(* CODESYS project Step.project
   Title: Step
   Version: 0.0.0.0
   Author: MustafaZahid

Project tree, tasks and I/O mapping:
  MyController : TM241C24T/U, Schneider Electric, order no. TM241C24T/U, version 4.0.6.18
    application Application
      task MAST (cyclic, interval 20 ms, priority 15, watchdog 100 ms x 1) calls POU
      global variables GVL
      program POU [LD]
    DI : Digital Inputs, Schneider Electric, version 4.0.6.18
        input  iwDI_IW0 : WORD  // IW0
        input  ibDI_IB1 : BYTE  // IB1
    DQ : Digital Outputs, Schneider Electric, version 4.0.6.18
        settings: Outputs Usage = 3
        output qwDQ_QW0 : WORD  // QW0
        output qbDQ_QB1 : BYTE  // QB1
    Counters : Counters, Schneider Electric, version 4.0.6.18
    Pulse_Generators : Pulse Generators, Schneider Electric, version 4.0.6.18
        settings: Instance name = 'Axis_1'; B output History = 'old=-1 new=1'; A output History = 'old=-1 new=0'; Temporary Instance name = 'Axis_1'
    Cartridge_1 : Cartridge, Schneider Electric, version 4.0.6.18
    IO_Bus : IO bus - TM3, Schneider Electric, version 4.0.6.18
    COM_Bus : COM bus, Schneider Electric, version 4.0.6.18
    Serial_Line_1 : Serial line, Schneider Electric, version 4.0.6.18
      SoMachine_Network_Manager : SoMachine-Network Manager, Schneider Electric, version 4.0.0.2
    Serial_Line_2 : Serial line, Schneider Electric, version 4.0.6.18
      Modbus_Manager : Modbus Manager, Schneider Electric, version 4.0.0.2
*)

// MyController/Application/GVL
VAR_GLOBAL
END_VAR

// MyController/Application/POU
PROGRAM POU
VAR
	MC_Power: MC_Power_PTO;
	MC_MoveVelocity: MC_MoveVelocity_PTO;
	MC_Reset: MC_Reset_PTO;
	Power: BOOL;
	Start: BOOL;
	Reset: BOOL;
	TON_0: TON;
	Speed: DINT;
	Dir: MC_DIRECTION;
END_VAR

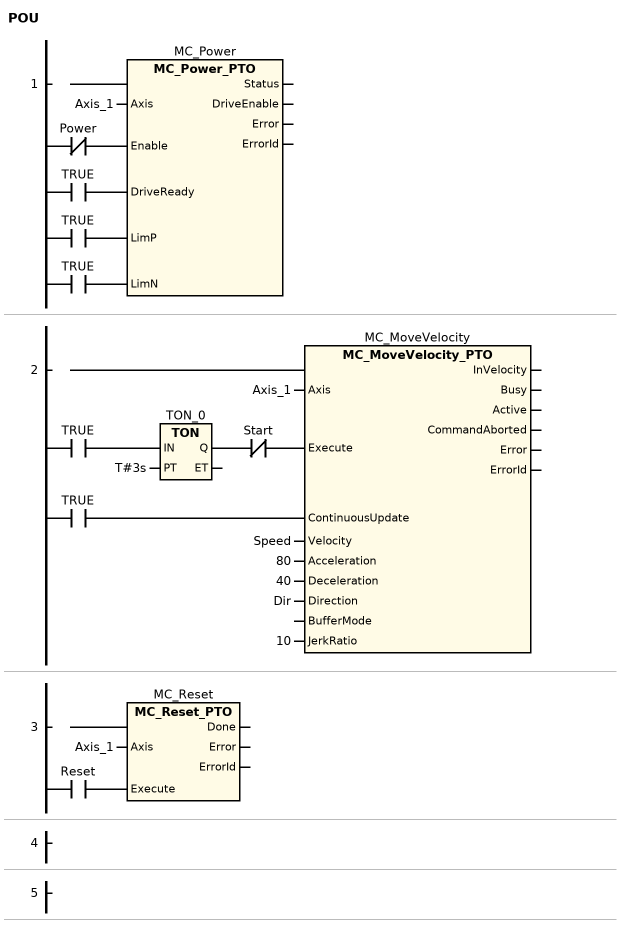
// NETWORK 1
MC_Power(Axis := Axis_1, Enable := NOT Power, DriveReady := TRUE, LimP := TRUE, LimN := TRUE); // MC_Power_PTO

// NETWORK 2
TON_0(IN := TRUE, PT := T#3s); // TON
MC_MoveVelocity(
    Axis := Axis_1,
    Execute := TON_0.Q AND NOT Start,
    ContinuousUpdate := TRUE,
    Velocity := Speed,
    Acceleration := 80,
    Deceleration := 40,
    Direction := Dir,
    JerkRatio := 10); // MC_MoveVelocity_PTO

// NETWORK 3
MC_Reset(Axis := Axis_1, Execute := Reset); // MC_Reset_PTO

// NETWORK 4

// NETWORK 5

END_PROGRAM
